TEXTLIST MachineMode
  0 = '電源OFF'
  1 = '初期化中'
  2 = '原点復帰中'
  3 = '初期化中'
  4 = '運転中'
  5 = 'サーボOFF中'
   = ''
END_TEXTLIST

(* stored: Version 1.1.0.1, ProductVersion 3.1.4024.12
   TextList MachineMode: Id {92b6ac52-ab5e-4326-a411-9cc194239317} *)
